FUNCTION F_LogLA9 
VAR_INPUT
	eLogLevel		: E_LogLevel;
	sLogger			: T_MaxString;
	sMessage		: T_MaxString;
	aArg1			: ANY;
	aArg2			: ANY;
	aArg3			: ANY;
	aArg4			: ANY;
	aArg5			: ANY;
	aArg6			: ANY;
	aArg7			: ANY;
	aArg8			: ANY;
	aArg9			: ANY;
END_VAR
VAR 
	aEmptyArg		: BYTE;
END_VAR

F_LogA(
	eLogLevel,
	sLogger,
	sMessage,
	4,
	aArg1,
	aArg2,
	aArg3,
	aArg4,
	aArg5,
	aArg6,
	aArg7,
	aArg8,
	aArg9,
	aEmptyArg
);

END_FUNCTION

(* stored: Version 1.1.0.1, ProductVersion 3.1.4024.0
   POU F_LogLA9: Id {c6db2f5c-acb8-423f-ad4a-09269318d8fe}, SpecialFunc None *)
